# EPICS substitutions: iocBoot/iocTomoScan_19BM/tomoScan.substitutions
# SAMPLE_X and SAMPLE_Y are the hexapod's X and Y axes.  The hexapod is
# installed at 7-BM today as 7bmbHXP: and is being moved here as-is; only the
# prefix and the controller IP change.  Its axes, from that IOC's
# motor.substitutions.automation1, are:
#
#     m1 Hexapod Z  mm   +/-27.5      m4 Hexapod A  deg  +/-7.5
#     m2 Hexapod X  mm   +/-30        m5 Hexapod B  deg  +/-7.5
#     m3 Hexapod Y  mm   0..500       m6 Hexapod C  deg  +/-15
#
# so replacing TODO_HEXAPOD with the new prefix is all that is needed.  Note
# Hexapod Y has a 0..500 mm range -- it is a lift rather than a fine
# translation, which is fine for moving a sample clear of the beam.
#
# SAMPLE_X / SAMPLE_Y are the translations UNDER the rotary, which tomoscan
# uses to move the sample clear of the beam for flat fields.  They are NOT the
# SampleTop X/Z pair on top of the rotary -- two Kohzu CYAT-070 stages, the
# centering stage, mounted here but not yet wired -- which co-rotates with
# theta and centres the sample on the rotation axis.  That pair is set by hand
# and has no tomoscan binding; do not rebind these macros to it once it is
# wired.
#
# 7-BM is not a useful reference for these: it binds them to 7bmb1:aero:m2 and
# :m1, two dedicated single-axis Ensembles that were commented out of
# 7bmb1's motor.aero.cmd in March 2026 ("not connected and slow down boot")
# while their records were left loaded, so 7-BM has been pointing at inert
# records ever since.
#
# The hexapod runs on an Aerotech Automation1 (10.54.107.77 today), a different
# controller from the Ensemble that drives the rotation, so 19-BM will end up
# with two Aerotech controllers.
#
# ROTATION is 19bmSoft:aero:m1, confirmed by the beamline 2026-09-19.  It is the
# Aerotech Ensemble air-bearing rotary stage, served by the 19bmSoft IOC on
# hounsfield.
#
# THE STAGE CANNOT BE MOVED YET.  The airflow interlock that makes rotating an
# air bearing safe is not wired up, so nothing should command this axis until
# the beamline says otherwise.  Binding the macro is safe -- tomoscan only
# reads the record until a scan is started -- but do not run a scan to "see
# what happens".
#
# CAMERA is the bare areaDetector IOC prefix; tomoscan.py appends "cam1:" itself.
# The 19-BM camera is a Vieworks VP-61MX (9568x6380, UInt16) on a Euresys
# Coaxlink grabber, driven by ADEuresys via ADGenICam.  Its IOC lives in
# /net/s19dserv/xorApps/epics/synApps_6_3/ioc/19bmVieworks and loads the
# standard commonPlugins.cmd set, so HDF1:, Pva1:, ROI1: and CB1: all exist.
file "$(TOP)/db/tomoScan.template"
{
pattern
{  P,       R,           CAMERA,          FILE_PLUGIN,          ROTATION,        SAMPLE_X,        SAMPLE_Y,           CLOSE_SHUTTER,        CLOSE_VALUE,          OPEN_SHUTTER,         OPEN_VALUE}
{19bm:, TomoScan:, 19bmVieworks:, 19bmVieworks:HDF1:, 19bmSoft:aero:m1, TODO_HEXAPOD:m2, TODO_HEXAPOD:m3, S19BM-PSS:FES:CloseEPICSC,       1,       S19BM-PSS:FES:OpenEPICSC,       1}
}

# For the Ensemble PSO_ENC_PER_ROTATION is a signed number containing the number of encoder pulses per rotation in positive dial coordinates
#
# These four values are NOT placeholders.  19-BM inherits the rotary stage and
# its Aerotech Ensemble controller from 7-BM intact, and all four are
# properties of that hardware rather than of where it is plugged in, so they
# carry over unchanged from iocTomoScan_7BM/tomoScan.substitutions.
#
# The one thing to re-verify after the stage is remounted is the SIGN of
# PSO_ENC_PER_ROTATION.  It is negative here because at 7-BM the encoder counts
# decrease as the dial position increases.  Remounting can reverse that.  Check
# it the way 32-ID-C documents: compare the signs of the rotation motor's .RVAL
# and .DRBV, which must agree for a positive value.
file "$(TOP)/db/tomoScan_PSO.template"
{
pattern
{  P,       R,      PSO_MODEL, PSO_PORT, PSO_AXIS_NAME, PSO_ENC_INPUT, PSO_ENC_PER_ROTATION}
{19bm:, TomoScan:,      0,     PSO_PORT,       A,             3,             -4096000.}
}

# Beamline-specific template.  Modeled on 7-BM rather than 32-ID-C because
# 32-ID-C's template carries an mctOptics prefix that 19-BM has no server for;
# the optics metadata records live in tomoScan_19BM.template itself.
#
# LINE is the GenICam TriggerSource the PSO output is wired to.  The Vieworks
# VP-61MX offers Software, UserOutput0, LinkTrigger0, Timer0Active and Line0.
# 19-BM has only the front-end shutter, bound through OPEN_SHUTTER /
# CLOSE_SHUTTER above; there are no fast-shutter macros because
# tomoScan_19BM.template defines no fast-shutter records.
#
# SHUTTER_STATUS reports whether the beam is BLOCKED: 1 = closed, 0 = open.
# That is the inverse of the PA:...:STA_?_SBS_OPEN_PL records used at 32-ID,
# and matches what 2-BM-B does with S02BM-PSS:SBS:BeamBlockingM.  The .VAL
# suffix follows 2-BM-B.
#
# BEAM_READY mirrors 2-BM-B, which uses S02BM-PSS:FES:FEEPSPermitM.
file "$(TOP)/db/tomoScan_19BM.template"
{
pattern
{  P,       R,             BEAM_READY,        READY_VALUE,          SHUTTER_STATUS,           LINE}
{19bm:, TomoScan:, S19BM-PSS:FES:FEEPSPermitM,      1,      S19BM-PSS:FES:BeamBlockingM.VAL, Line0}
}
